TYPE ST_Control :
STRUCT
	bReset:		BOOL;
	bSwitch:	BOOL;
END_STRUCT
END_TYPE

(* stored: Version 1.1.0.1, ProductVersion 3.1.4024.12
   DUT ST_Control: Id {cc30844c-3d8d-43d2-9971-8c9e1035a665} *)
